{attribute addProperty BoxType "ER6002-0002-0021"}
{attribute addProperty Id "COM_TxPDO_Map_Inputs_ChannelAT %I*ARRAY[0..23] OF COM_TxPDO_Map_Inputs_Channel_4EE430B6384480COM_RxPDO_Map_Outputs_ChannelAT %Q*ARRAY[0..23] OF COM_RxPDO_Map_Outputs_Channel_CEA6CFDD384480WcStateAT %I*WcState_98A4DF7520.250InfoDataAT %I*InfoData_BC63D37F80100"}
{attribute addProperty CRC "2888717740"}
{attribute addProperty SizeInBites "850"}
{attribute addProperty SizeInBytes "106.25"}
TYPE ER6002_320F021A :
STRUCT
	{attribute addProperty Name "COM_TxPDO_Map_Inputs_Channel"}
	COM_TxPDO_Map_Inputs_Channel : ARRAY[0..23] OF COM_TxPDO_Map_Inputs_Channel_4EE430B6;
	{attribute addProperty Name "COM_RxPDO_Map_Outputs_Channel"}
	COM_RxPDO_Map_Outputs_Channel : ARRAY[0..23] OF COM_RxPDO_Map_Outputs_Channel_CEA6CFDD;
	{attribute addProperty Name "WcState"}
	WcState : WcState_98A4DF75;
	{attribute addProperty Name "InfoData"}
	InfoData : InfoData_BC63D37F;
END_STRUCT
END_TYPE

(* stored: Version 1.2.0.0, ProductVersion 3.1.4024.9
   DUT ER6002_320F021A: Id {0a0f90f8-63ed-49b8-9e97-cc8cfee8f9fa} *)
